KUKA KRL program: f_fraes3.src, f_fraes3.dat

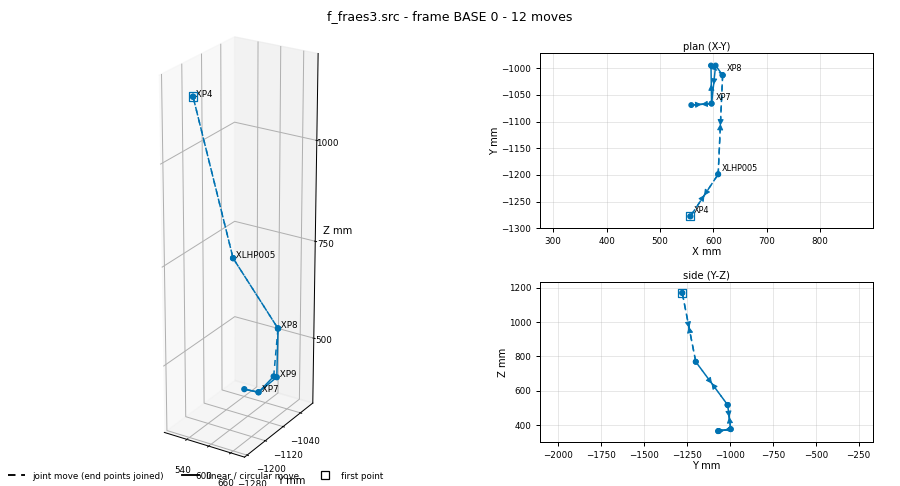
[picture p0: tool path of f_fraes3.src in frame BASE 0, 12 of 12 moves have a stored position in this frame; points joined in program order, loops and branches not executed]
--- f_fraes3.src ---
&ACCESS RVO7
&REL 2
&COMMENT Fresa C2
&PARAM DISKPATH = KRC:\R1\Program
&PARAM TEMPLATE = C:\KRC\Roboter\Template\vorgabe
&PARAM EDITMASK = *
DEF f_fraes3( )
;FOLD INI
   ;FOLD BASISTECH INI
      GLOBAL INTERRUPT DECL 3 WHEN $STOPMESS==TRUE DO IR_STOPM ( )
      INTERRUPT ON 3
      BAS (#INITMOV,0 )
   ;ENDFOLD (BASISTECH INI)
   ;FOLD SPOTTECH INI
      USERSPOT(#INIT)
   ;ENDFOLD (SPOTTECH INI)
   ;FOLD GRIPPERTECH INI
      USER_GRP(0,DUMMY,DUMMY,GDEFAULT)
   ;ENDFOLD (GRIPPERTECH INI)
   ;FOLD USER INI
      ;Make your modifications here

   ;ENDFOLD (USER INI)
;ENDFOLD (INI)

; Estacao P13.060 - Robo R2
; Programa: Fresa C2
; Caracterização dos meios de produção:
; 02/09/2014 09:15 Changes by KUKA Roboter do Brasil

chk_w3_wechs_ok () ;check c2

;FOLD PTP P4 Vel=80 % PDAT6 Tool[3]:Pinca C2 Base[0];%{PE}%R 8.2.20,%MKUKATPBASIS,%CMOVE,%VPTP,%P 1:PTP, 2:P4, 3:, 5:80, 7:PDAT6
$BWDSTART=FALSE
PDAT_ACT=PPDAT6
FDAT_ACT=FP4
BAS(#PTP_PARAMS,80)
PTP XP4
;ENDFOLD
;FOLD PTP LHP005 CONT Vel=60 % PDAT2 Tool[3]:Pinca C2 Base[0];%{PE}%R 8.2.20,%MKUKATPBASIS,%CMOVE,%VPTP,%P 1:PTP, 2:LHP005, 3:C_DIS, 5:60, 7:PDAT2
$BWDSTART=FALSE
PDAT_ACT=PPDAT2
FDAT_ACT=FLHP005
BAS(#PTP_PARAMS,60)
PTP XLHP005 C_DIS
;ENDFOLD
;FOLD PTP P8 Vel=60 % PDAT11 Tool[3]:Pinca C2 Base[0];%{PE}%R 8.2.20,%MKUKATPBASIS,%CMOVE,%VPTP,%P 1:PTP, 2:P8, 3:, 5:60, 7:PDAT11
$BWDSTART=FALSE
PDAT_ACT=PPDAT11
FDAT_ACT=FP8
BAS(#PTP_PARAMS,60)
PTP XP8
;ENDFOLD
;FOLD LIN P9 Vel=0.3 m/s CPDAT2 Tool[3]:Pinca C2 Base[0];%{PE}%R 8.2.20,%MKUKATPBASIS,%CMOVE,%VLIN,%P 1:LIN, 2:P9, 3:, 5:0.3, 7:CPDAT2
$BWDSTART=FALSE
LDAT_ACT=LCPDAT2
FDAT_ACT=FP9
BAS(#CP_PARAMS,0.3)
LIN XP9
;ENDFOLD
;FOLD LIN P7 Vel=0.3 m/s CPDAT1 Tool[3]:Pinca C2 Base[0];%{PE}%R 8.2.20,%MKUKATPBASIS,%CMOVE,%VLIN,%P 1:LIN, 2:P7, 3:, 5:0.3, 7:CPDAT1
$BWDSTART=FALSE
LDAT_ACT=LCPDAT1
FDAT_ACT=FP7
BAS(#CP_PARAMS,0.3)
LIN XP7
;ENDFOLD

;FOLD ; PONTO DE FRESAGEM;%{PE}%R 4.1.16,%MKUKATPBASIS,%CCOMMENT,%VNORMAL,%P 2:PONTO DE FRESAGEM
;ENDFOLD
;FOLD TIP.LIN_ Dress2, Spot Gun 2 , RETR open , Tool[3], Base[0], EXT.TCP=FALSE;%{PE}%MKUKATPUSER
FDAT_ACT=FDress2
BAS(#FRAMES)
LIN  XDress2
S_ACT.GUN=2
S_ACT.RETR=#opn
S_READY=FALSE
USERSPOT (#DRESS,S_ACT )
WAIT FOR  S_READY
;ENDFOLD

;FOLD LIN P1 Vel=0.3 m/s CPDAT4 Tool[3]:Pinca C2 Base[0];%{PE}%R 8.2.20,%MKUKATPBASIS,%CMOVE,%VLIN,%P 1:LIN, 2:P1, 3:, 5:0.3, 7:CPDAT4
$BWDSTART=FALSE
LDAT_ACT=LCPDAT4
FDAT_ACT=FP1
BAS(#CP_PARAMS,0.3)
LIN XP1
;ENDFOLD
;FOLD LIN P11 Vel=0.3 m/s CPDAT3 Tool[3]:Pinca C2 Base[0];%{PE}%R 8.2.20,%MKUKATPBASIS,%CMOVE,%VLIN,%P 1:LIN, 2:P11, 3:, 5:0.3, 7:CPDAT3
$BWDSTART=FALSE
LDAT_ACT=LCPDAT3
FDAT_ACT=FP11
BAS(#CP_PARAMS,0.3)
LIN XP11
;ENDFOLD
;FOLD PTP LHP025 Vel=60 % PDAT7 Tool[3]:Pinca C2 Base[0];%{PE}%R 8.2.20,%MKUKATPBASIS,%CMOVE,%VPTP,%P 1:PTP, 2:LHP025, 3:, 5:60, 7:PDAT7
$BWDSTART=FALSE
PDAT_ACT=PPDAT7
FDAT_ACT=FLHP025
BAS(#PTP_PARAMS,60)
PTP XLHP025
;ENDFOLD

;FOLD PTP pTEST_WELD PDAT5 SPOT Gun=2 RETR OPN PgNo1=252 ACTIVE=1 NORMAL Tool[3]:Pinca C2 Base[0];%{PE}%R 8.2.2,%MKUKATPSPOT,%CSPOT,%VPTP,%P 1:PTP, 2:pTEST_WELD, 3:, 5:60, 7:PDAT5, 10:2, 12:#FIRST, 14:#OPN, 16:252, 18:1, 20:0, 22:0, 24:1, 25:NORMAL
$BWDSTART=FALSE
PDAT_ACT=PPDAT5
FDAT_ACT=FpTEST_WELD
BAS(#PTP_PARAMS,PPDAT5.VEL)
S_ACT.GUN=2
S_ACT.PAIR=SDEFAULT.PAIR
S_ACT.RETR=#OPN
S_ACT.CLO_TM=1
S_ACT.PGNO1=252
S_ACT.PGNO2=SDEFAULT.PGNO2
S_ACT.PRESS1=SDEFAULT.PRESS1
S_ACT.PRESS2=SDEFAULT.PRESS2
S_READY=FALSE
PTP XpTEST_WELD
USERSPOT(#SPOT, S_ACT)
WAIT FOR S_READY

;ENDFOLD

;FOLD PTP P2 CONT Vel=60 % PDAT4 Tool[3]:Pinca C2 Base[0];%{PE}%R 8.2.20,%MKUKATPBASIS,%CMOVE,%VPTP,%P 1:PTP, 2:P2, 3:C_DIS, 5:60, 7:PDAT4
$BWDSTART=FALSE
PDAT_ACT=PPDAT4
FDAT_ACT=FP2
BAS(#PTP_PARAMS,60)
PTP XP2 C_DIS
;ENDFOLD
;FOLD PTP P3 Vel=100 % PDAT9 Tool[3]:Pinca C2 Base[0];%{PE}%R 8.2.20,%MKUKATPBASIS,%CMOVE,%VPTP,%P 1:PTP, 2:P3, 3:, 5:100, 7:PDAT9
$BWDSTART=FALSE
PDAT_ACT=PPDAT9
FDAT_ACT=FP3
BAS(#PTP_PARAMS,100)
PTP XP3
;ENDFOLD


END

--- f_fraes3.dat ---
&ACCESS RVO7
&REL 2
&COMMENT Fresa C2
&PARAM DISKPATH = KRC:\R1\Program
&PARAM TEMPLATE = C:\KRC\Roboter\Template\vorgabe
&PARAM EDITMASK = *
DEFDAT  f_fraes3
;FOLD EXTERNAL DECLARATIONS;%{PE}%MKUKATPBASIS,%CEXT,%VCOMMON,%P
;FOLD GRIPPERTECH EXT
EXT  H50 (INT  :IN,INT  :IN,INT  :IN,GRP_TYP  :IN )
;ENDFOLD (GRIPPERTECH EXT)
;FOLD SPOTTECH EXT
EXT  USERSPOT (S_COMMAND  :IN,SPOT_TYPE  :IN )
;ENDFOLD (SPOTTECH EXT)
;FOLD BASISTECH EXT;%{PE}%MKUKATPBASIS,%CEXT,%VEXT,%P
EXT  BAS (BAS_COMMAND  :IN,REAL  :IN )
DECL INT SUCCESS
;ENDFOLD (BASISTECH EXT)
;FOLD USER EXT;%{E}%MKUKATPUSER,%CEXT,%VEXT,%P
;Make your modifications here

;ENDFOLD (USER EXT)
;ENDFOLD (EXTERNAL DECLARATIONS)

DECL PDAT PPDAT2={VEL 80.0,ACC 100.0,APO_DIST 20.0,APO_MODE #CDIS}
DECL E6POS XLHP025={X 617.337891,Y -1013.08301,Z 517.776917,A -87.1397629,B 11.1259899,C 91.5856628,S 18,T 34,E1 0.0,E2 0.0,E3 0.0,E4 0.0,E5 0.0,E6 0.0}
DECL FDAT FLHP025={TOOL_NO 3,BASE_NO 0,IPO_FRAME #BASE,TQ_STATE FALSE}
DECL PDAT PPDAT7={VEL 100.0,ACC 100.0,APO_DIST 10.0,APO_MODE #CDIS}
DECL E6POS XLHP020={X 638.080872,Y -1075.26794,Z 367.941803,A -89.7975464,B 3.68088388,C 91.0812836,S 18,T 34,E1 0.0,E2 0.0,E3 0.0,E4 0.0,E5 0.0,E6 0.0}
DECL FDAT FLHP020={TOOL_NO 3,BASE_NO 0,IPO_FRAME #BASE,TQ_STATE FALSE}
DECL LDAT LCPDAT16={VEL 2.0,ACC 100.0,APO_DIST 5.0,APO_FAC 50.0}
DECL E6POS XPTEST_WELD={X 617.334717,Y -1013.073,Z 517.778809,A -87.139473,B 11.1263399,C 91.5856781,S 18,T 34,E1 0.0,E2 0.0,E3 0.0,E4 0.0,E5 0.0,E6 0.0}
DECL FDAT FpTEST_WELD={TOOL_NO 3,BASE_NO 0,IPO_FRAME #BASE,TQ_STATE FALSE}
DECL PDAT PPDAT10={VEL 100.0,ACC 100.0,APO_DIST 100.0}
DECL E6POS XLHP005={X 608.984009,Y -1198.71594,Z 769.078979,A -90.0554886,B 6.36685991,C 91.3043594,S 18,T 34,E1 0.0,E2 0.0,E3 0.0,E4 0.0,E5 0.0,E6 0.0}
DECL FDAT FLHP005={TOOL_NO 3,BASE_NO 0,IPO_FRAME #BASE,TQ_STATE FALSE}
DECL BASIS_SUGG_T LAST_BASIS={POINT1[] "P3                      ",POINT2[] "P3                      ",CP_PARAMS[] "CPDAT0                  ",PTP_PARAMS[] "PDAT9                   ",CONT[] "                        ",CP_VEL[] "0.3                     ",PTP_VEL[] "100                     ",SYNC_PARAMS[] "SYNCDAT                 ",SPL_NAME[] "S0                      "}
DECL E6POS XP2={X 608.984009,Y -1198.71594,Z 769.078979,A -90.0554886,B 6.36685991,C 91.3043594,S 18,T 34,E1 0.0,E2 0.0,E3 0.0,E4 0.0,E5 0.0,E6 0.0}
DECL FDAT FP2={TOOL_NO 3,BASE_NO 0,IPO_FRAME #BASE,POINT2[] " ",TQ_STATE FALSE}
DECL PDAT PPDAT4={VEL 100.0,ACC 100.0,APO_DIST 50.0,APO_MODE #CDIS,GEAR_JERK 50.0}
DECL E6POS XP4={X 556.892395,Y -1277.56494,Z 1169.94202,A -90.058197,B -16.1502991,C 90.6416702,S 18,T 42,E1 0.0,E2 0.0,E3 0.0,E4 0.0,E5 0.0,E6 0.0}
DECL FDAT FP4={TOOL_NO 3,BASE_NO 0,IPO_FRAME #BASE,POINT2[] " ",TQ_STATE FALSE}
DECL PDAT PPDAT6={VEL 100.0,ACC 100.0,APO_DIST 10.0,APO_MODE #CDIS,GEAR_JERK 50.0}
DECL E6POS XP7={X 596.642273,Y -1066.30103,Z 365.804688,A -89.7720184,B 5.3642149,C 91.0782166,S 18,T 34,E1 0.0,E2 0.0,E3 0.0,E4 0.0,E5 0.0,E6 0.0}
DECL FDAT FP7={TOOL_NO 3,BASE_NO 0,IPO_FRAME #BASE,POINT2[] " ",TQ_STATE FALSE}
DECL LDAT LCPDAT1={VEL 2.0,ACC 100.0,APO_DIST 100.0,APO_FAC 50.0,AXIS_VEL 100.0,AXIS_ACC 100.0,ORI_TYP #VAR,CIRC_TYP #BASE,JERK_FAC 50.0,GEAR_JERK 50.0,EXAX_IGN 0}
DECL FDAT FDress2={TOOL_NO 3,BASE_NO 0,IPO_FRAME #BASE}
DECL E6POS XDress2={X 558.609619,Y -1069.10596,Z 364.770599,A -89.7720871,B 5.36627102,C 91.0785065,S 18,T 34,E1 0.0,E2 0.0,E3 0.0,E4 0.0,E5 0.0,E6 0.0}
DECL E6POS XP8={X 617.341614,Y -1013.08899,Z 517.776489,A -87.13974,B 11.1255798,C 91.5857773,S 18,T 34,E1 0.0,E2 0.0,E3 0.0,E4 0.0,E5 0.0,E6 0.0}
DECL FDAT FP8={TOOL_NO 3,BASE_NO 0,IPO_FRAME #BASE,POINT2[] " ",TQ_STATE FALSE}
DECL PDAT PPDAT11={VEL 100.0,ACC 100.0,APO_DIST 100.0,GEAR_JERK 50.0}
DECL E6POS XP9={X 604.204773,Y -995.019592,Z 376.719513,A -89.7470627,B 7.071383,C 91.0780334,S 18,T 34,E1 0.0,E2 0.0,E3 0.0,E4 0.0,E5 0.0,E6 0.0}
DECL FDAT FP9={TOOL_NO 3,BASE_NO 0,IPO_FRAME #BASE,POINT2[] " ",TQ_STATE FALSE}
DECL LDAT LCPDAT2={VEL 2.0,ACC 100.0,APO_DIST 100.0,APO_FAC 50.0,AXIS_VEL 100.0,AXIS_ACC 100.0,ORI_TYP #VAR,CIRC_TYP #BASE,JERK_FAC 50.0,GEAR_JERK 50.0,EXAX_IGN 0}
DECL E6POS XP11={X 595.499817,Y -995.021484,Z 376.545593,A -89.7470474,B 7.07201576,C 91.0777588,S 18,T 34,E1 0.0,E2 0.0,E3 0.0,E4 0.0,E5 0.0,E6 0.0}
DECL FDAT FP11={TOOL_NO 3,BASE_NO 0,IPO_FRAME #BASE,POINT2[] " ",TQ_STATE FALSE}
DECL LDAT LCPDAT3={VEL 2.0,ACC 100.0,APO_DIST 100.0,APO_FAC 50.0,AXIS_VEL 100.0,AXIS_ACC 100.0,ORI_TYP #VAR,CIRC_TYP #BASE,JERK_FAC 50.0,GEAR_JERK 50.0,EXAX_IGN 0}
DECL E6POS XP1={X 596.638306,Y -1066.29504,Z 365.808502,A -89.7720337,B 5.36458492,C 91.0780869,S 18,T 34,E1 0.0,E2 0.0,E3 0.0,E4 0.0,E5 0.0,E6 0.0}
DECL FDAT FP1={TOOL_NO 3,BASE_NO 0,IPO_FRAME #BASE,POINT2[] " ",TQ_STATE FALSE}
DECL PDAT PPDAT1={VEL 100.0,ACC 100.0,APO_DIST 100.0,GEAR_JERK 50.0}
DECL LDAT LCPDAT4={VEL 2.0,ACC 100.0,APO_DIST 100.0,APO_FAC 50.0,AXIS_VEL 100.0,AXIS_ACC 100.0,ORI_TYP #VAR,CIRC_TYP #BASE,JERK_FAC 50.0,GEAR_JERK 50.0,EXAX_IGN 0}
DECL SPOT_SUGG_T LAST_SPOT={GUN[] " 1                      ",RETR_CMD[] "#OPN                    ",CHOISE[] "#FIRST                  ",CLO_TM[] "0                       ",PGNO1[] " 1                      ",PRESS1[] "0                       ",PGNO2[] " 1                      ",PRESS2[] "0                       ",SPOT_PARAMS[] "NORMAL                  "}
DECL PDAT PPDAT3={VEL 100.0,ACC 100.0,APO_DIST 100.0}
DECL SPOT_TYPE SNORMAL={GUN 1,PAIR #FIRST,RETR #OPN,CLO_TM 0,PGNO1 1,PRESS1 0.0,PGNO2 0,PRESS2 0.0}
DECL PDAT PPDAT5={VEL 100.0,ACC 100.0,APO_DIST 100.0}
DECL PDAT PPDAT8={VEL 100.0,ACC 100.0,APO_DIST 100.0}
DECL E6POS XP3={X 556.879578,Y -1277.56604,Z 1169.93298,A -90.0581284,B -16.1495399,C 90.6412506,S 18,T 42,E1 0.0,E2 0.0,E3 0.0,E4 0.0,E5 0.0,E6 0.0}
DECL FDAT FP3={TOOL_NO 3,BASE_NO 0,IPO_FRAME #BASE,POINT2[] " ",TQ_STATE FALSE}
DECL PDAT PPDAT9={VEL 100.0,ACC 100.0,APO_DIST 100.0,APO_MODE #CDIS,GEAR_JERK 50.0}
ENDDAT
